FUNCTION_BLOCK FB_SubSubNestedView EXTENDS FB_SubNestedView
VAR_INPUT CONSTANT
	SubX		: FB_SubNestedView		:= (iParent:=THIS^);
END_VAR

SUPER^();

SubX();

END_FUNCTION_BLOCK

(* stored: Version 1.1.0.1, ProductVersion 3.1.4024.5
   POU FB_SubSubNestedView: Id {4483bd18-9ab6-41f9-abb3-e977c7290f61}, SpecialFunc None *)
